Fanuc TP program (LS listing): _VAC_ON.LS

/PROG  _VAC_ON
/ATTR
OWNER		= MNEDITOR;
COMMENT		= "Vac SubRoutine";
PROG_SIZE	= 526;
CREATE		= DATE 23-09-05  TIME 15:42:24;
MODIFIED	= DATE 23-09-05  TIME 15:57:20;
FILE_NAME	= VACON;
VERSION		= 0;
LINE_COUNT	= 10;
MEMORY_SIZE	= 858;
PROTECT		= READ_WRITE;
TCD:  STACK_SIZE	= 0,
      TASK_PRIORITY	= 50,
      TIME_SLICE	= 0,
      BUSY_LAMP_OFF	= 0,
      ABORT_REQUEST	= 0,
      PAUSE_REQUEST	= 0;
DEFAULT_GROUP	= 1,*,*,*,*;
CONTROL_CODE	= 00000000 00000000;
LOCAL_REGISTERS	= 0,0,0;
/APPL
/APPL

AUTO_SINGULARITY_HEADER;
  ENABLE_SINGULARITY_AVOIDANCE   : FALSE;

PLTZ_MODE_HEADER;
 PLTZ_MODE_ENABLE   : FALSE;
 J4TURN  : ZERORAD;
 ORIENT  : DOWNWARDS;
/MN
   1:  !---------------------------- ;
   2:  !  CRX25 Palletizing Demo     ;
   3:  !   Vacuum SubRoutine         ;
   4:  !                             ;
   5:  !  BY: JDM                    ;
   6:  !  DATE: 8.31.2023            ;
   7:  !---------------------------- ;
   8:  DO[102:BLOW_OFF]=OFF ;
   9:  DO[101:VAC_ON]=ON ;
  10:  WAIT    .50(sec) ;
/POS
/END
